# EPICS autosave request: dxp/tags/R3-0/dxpApp/Db/dxpSystem_settings.req
$(P)PollTime
$(P)NumSCAs
$(P)SaveSystemFile
